// TIA Portal V16 export
// export: Created 2024-06-17T18:37:12.7801223Z, ExportSetting WithDefaults, DisplayName Totally Integrated Automation Portal, DisplayVersion V16, DisplayName TIA Portal Version Control Interface, DisplayVersion V16, DisplayName TIA Portal Openness, DisplayVersion V16, DisplayName STEP 7 Professional, DisplayVersion V16, DisplayName STEP 7 Safety, DisplayVersion V16, DisplayName WinCC Advanced, DisplayVersion V16
TYPE "Axis.RB.Di_PLC.Do"
TITLE = Saídas para robô
// stored: IsFailsafeCompliant false
   STRUCT
      "RB.Gi_PLC.Go_NumProg" : Int;   // Numero Programa
      "RB.Di_PLC.Do16_IniciaProcesso" : Bool;   // Autoriza Número de Programa Processo
      "RB.Di_PLC.Do17_ProgramaOK" : Bool;   // Confirma numero de programa
      "RB.Di_PLC.Do18_MotorOn" : Bool;   // Liga Motores
      "RB.Di_PLC.Do19_MotorOff" : Bool;   // Desliga Motores
      "RB.Di_PLC.Do20_StartRob" : Bool;   // Partida Execução Programa (Play)
      "RB.Di_PLC.Do21_StopRob" : Bool;   // Pausa execução programa (Stop)
      "RB.Di_PLC.Do22_Reserva" : Bool;   // Reserva
      "RB.Di_PLC.Do23_Reserva" : Bool;   // Reserva
      "RB.Di_PLC.Do24_CicloVazio" : Bool;   // Modo Ciclo Vazio
      "RB.Di_PLC.Do25_SolicitaParada" : Bool;   // Pedido de Parada para Entrada na Célula
      "RB.Di_PLC.Do26_CancelaTrabalho" : Bool;   // Aborta uma Trajetória Não Iniciada
      "RB.Di_PLC.Do27_ResetFalha" : Bool;   // Reset Falha
      "RB.Di_PLC.Do28_RetornaManutencao" : Bool;   // Pedido de Retorno da Posição de Manutenção
      "RB.Di_PLC.Do29_RetornaCalibracao" : Bool;   // Pedido de Retorno da Posição de Calibração
      "RB.Di_PLC.Do30_RetornaSincronismo" : Bool;   // Pedido de Retorno da Posição de Sincronismo
      "RB.Di_PLC.Do31_Reserva" : Bool;   // Reserva
      "RB.Di_PLC.Do32_Pressao_Ar_OK" : Bool;   // Pressão de Ar OK
      "RB.Di_PLC.Do33_Reserva" : Bool;   // Reserva
      "RB.Di_PLC.Do34_Reserva" : Bool;   // Reserva
      "RB.Di_PLC.Do35_Reserva" : Bool;   // Reserva
      "RB.Di_PLC.Do36_Reserva" : Bool;   // Reserva
      "RB.Di_PLC.Do37_Reserva" : Bool;   // Reserva
      "RB.Di_PLC.Do38_Reserva" : Bool;   // Reserva
      "RB.Di_PLC.Do39_Reserva" : Bool;   // Reserva
      "RB.Di_PLC.Do40_Reserva" : Bool;   // Reserva
      "RB.Di_PLC.Do41_Reserva" : Bool;   // Reserva
      "RB.Di_PLC.Do42_Reserva" : Bool;   // Reserva
      "RB.Di_PLC.Do43_Reserva" : Bool;   // Reserva
      "RB.Di_PLC.Do44_Reserva" : Bool;   // Reserva
      "RB.Di_PLC.Do45_Reserva" : Bool;   // Reserva
      "RB.Di_PLC.Do46_Reserva" : Bool;   // Reserva
      "RB.Di_PLC.Do47_Reserva" : Bool;   // Reserva
      "RB.Di_PLC.Do48_Reserva" : Bool;   // Reserva
      "RB.Di_PLC.Do49_Reserva" : Bool;   // Reserva
      "RB.Di_PLC.Do50_Reserva" : Bool;   // Reserva
      "RB.Di_PLC.Do51_Reserva" : Bool;   // Reserva
      "RB.Di_PLC.Do52_Reserva" : Bool;   // Reserva
      "RB.Di_PLC.Do53_Reserva" : Bool;   // Reserva
      "RB.Di_PLC.Do54_Reserva" : Bool;   // Reserva
      "RB.Di_PLC.Do55_Reserva" : Bool;   // Reserva
      "RB.Di_PLC.Do56_Aut.Trabalho_1" : Bool;   // Autoriza Trabalho 1
      "RB.Di_PLC.Do57_Aut.Trabalho_2" : Bool;   // Autoriza Trabalho 2
      "RB.Di_PLC.Do58_Aut.Trabalho_3" : Bool;   // Autoriza Trabalho 3
      "RB.Di_PLC.Do59_Aut.Trabalho_4" : Bool;   // Autoriza Trabalho 4
      "RB.Di_PLC.Do60_Aut.Trabalho_5" : Bool;   // Autoriza Trabalho 5
      "RB.Di_PLC.Do61_Aut.Trabalho_6" : Bool;   // Autoriza Trabalho 6
      "RB.Di_PLC.Do62_Aut.Trabalho_7" : Bool;   // Autoriza Trabalho 7
      "RB.Di_PLC.Do63_Aut.Trabalho_8" : Bool;   // Autoriza Trabalho 8
      "RB.Di_PLC.Do64_Aut.Trabalho_9" : Bool;   // Autoriza Trabalho 9
      "RB.Di_PLC.Do65_Aut.Trabalho_10" : Bool;   // Autoriza Trabalho 10
      "RB.Di_PLC.Do66_Aut.Trabalho_11" : Bool;   // Autoriza Trabalho 11
      "RB.Di_PLC.Do67_Aut.Trabalho_12" : Bool;   // Autoriza Trabalho 12
      "RB.Di_PLC.Do68_Aut.Trabalho_13" : Bool;   // Autoriza Trabalho 13
      "RB.Di_PLC.Do69_Aut.Trabalho_14" : Bool;   // Autoriza Trabalho 14
      "RB.Di_PLC.Do70_Aut.Trabalho_15" : Bool;   // Autoriza Trabalho 15
      "RB.Di_PLC.Do71_Aut.Trabalho_16" : Bool;   // Autoriza Trabalho 16
      "RB.Di_PLC.Do72_Aut.Trabalho_17" : Bool;   // Autoriza Trabalho 17
      "RB.Di_PLC.Do73_Aut.Trabalho_18" : Bool;   // Autoriza Trabalho 18
      "RB.Di_PLC.Do74_Aut.Trabalho_19" : Bool;   // Autoriza Trabalho 19
      "RB.Di_PLC.Do75_Aut.Trabalho_20" : Bool;   // Autoriza Trabalho 20
      "RB.Di_PLC.Do76_Aut.Trabalho_21" : Bool;   // Autoriza Trabalho 21
      "RB.Di_PLC.Do77_Aut.Trabalho_22" : Bool;   // Autoriza Trabalho 22
      "RB.Di_PLC.Do78_Aut.Trabalho_23" : Bool;   // Autoriza Trabalho 23
      "RB.Di_PLC.Do79_Aut.Trabalho_24" : Bool;   // Autoriza Trabalho 24
      "RB.Di_PLC.Do80_Aut.Trabalho_25" : Bool;   // Autoriza Trabalho 25
      "RB.Di_PLC.Do81_Aut.Trabalho_26" : Bool;   // Autoriza Trabalho 26
      "RB.Di_PLC.Do82_Aut.Trabalho_27" : Bool;   // Autoriza Trabalho 27
      "RB.Di_PLC.Do83_Aut.Trabalho_28" : Bool;   // Autoriza Trabalho 28
      "RB.Di_PLC.Do84_Aut.Trabalho_29" : Bool;   // Autoriza Trabalho 29
      "RB.Di_PLC.Do85_Aut.Trabalho_30" : Bool;   // Autoriza Trabalho 30
      "RB.Di_PLC.Do86_Aut.Trabalho_31" : Bool;   // Autoriza Trabalho 31
      "RB.Di_PLC.Do87_Aut.Trabalho_32" : Bool;   // Autoriza Trabalho 32
      "RB.Di_PLC.Do88_Aut.Intertravamento_1" : Bool;   // Autoriza Acesso Área Intertravamento 1
      "RB.Di_PLC.Do89_Aut.Intertravamento_2" : Bool;   // Autoriza Acesso Área Intertravamento 2
      "RB.Di_PLC.Do90_Aut.Intertravamento_3" : Bool;   // Autoriza Acesso Área Intertravamento 3
      "RB.Di_PLC.Do91_Aut.Intertravamento_4" : Bool;   // Autoriza Acesso Área Intertravamento 4
      "RB.Di_PLC.Do92_Aut.Intertravamento_5" : Bool;   // Autoriza Acesso Área Intertravamento 5
      "RB.Di_PLC.Do93_Aut.Intertravamento_6" : Bool;   // Autoriza Acesso Área Intertravamento 6
      "RB.Di_PLC.Do94_Aut.Intertravamento_7" : Bool;   // Autoriza Acesso Área Intertravamento 7
      "RB.Di_PLC.Do95_Aut.Intertravamento_8" : Bool;   // Autoriza Acesso Área Intertravamento 8
      "RB.Di_PLC.Do96_Aut.Intertravamento_9" : Bool;   // Autoriza Acesso Área Intertravamento 9
      "RB.Di_PLC.Do97_Aut.Intertravamento_10" : Bool;   // Autoriza Acesso Área Intertravamento 10
      "RB.Di_PLC.Do98_Aut.Intertravamento_11" : Bool;   // Autoriza Acesso Área Intertravamento 11
      "RB.Di_PLC.Do99_Aut.Intertravamento_12" : Bool;   // Autoriza Acesso Área Intertravamento 12
      "RB.Di_PLC.Do100_Aut.Intertravamento_13" : Bool;   // Autoriza Acesso Área Intertravamento 13
      "RB.Di_PLC.Do101_Aut.Intertravamento_14" : Bool;   // Autoriza Acesso Área Intertravamento 14
      "RB.Di_PLC.Do102_Aut.Intertravamento_15" : Bool;   // Autoriza Acesso Área Intertravamento 15
      "RB.Di_PLC.Do103_Aut.Intertravamento_16" : Bool;   // Autoriza Acesso Área Intertravamento 16
      "RB.Di_PLC.Do104_Aut.Intertravamento_17" : Bool;   // Autoriza Acesso Área Intertravamento 17
      "RB.Di_PLC.Do105_Aut.Intertravamento_18" : Bool;   // Autoriza Acesso Área Intertravamento 18
      "RB.Di_PLC.Do106_Aut.Intertravamento_19" : Bool;   // Autoriza Acesso Área Intertravamento 19
      "RB.Di_PLC.Do107_Aut.Intertravamento_20" : Bool;   // Autoriza Acesso Área Intertravamento 20
      "RB.Di_PLC.Do108_Aut.Intertravamento_21" : Bool;   // Autoriza Acesso Área Intertravamento 21
      "RB.Di_PLC.Do109_Aut.Intertravamento_22" : Bool;   // Autoriza Acesso Área Intertravamento 22
      "RB.Di_PLC.Do110_Aut.Intertravamento_23" : Bool;   // Autoriza Acesso Área Intertravamento 23
      "RB.Di_PLC.Do111_Aut.Intertravamento_24" : Bool;   // Autoriza Acesso Área Intertravamento 24
      "RB.Di_PLC.Do112_Aut.Intertravamento_25" : Bool;   // Autoriza Acesso Área Intertravamento 25
      "RB.Di_PLC.Do113_Aut.Intertravamento_26" : Bool;   // Autoriza Acesso Área Intertravamento 26
      "RB.Di_PLC.Do114_Aut.Intertravamento_27" : Bool;   // Autoriza Acesso Área Intertravamento 27
      "RB.Di_PLC.Do115_Aut.Intertravamento_28" : Bool;   // Autoriza Acesso Área Intertravamento 28
      "RB.Di_PLC.Do116_Aut.Intertravamento_29" : Bool;   // Autoriza Acesso Área Intertravamento 29
      "RB.Di_PLC.Do117_Aut.Intertravamento_30" : Bool;   // Autoriza Acesso Área Intertravamento 30
      "RB.Di_PLC.Do118_Aut.Intertravamento_31" : Bool;   // Autoriza Acesso Área Intertravamento 31
      "RB.Di_PLC.Do119_Aut.Intertravamento_32" : Bool;   // Autoriza Acesso Área Intertravamento 32
      "RB.Di_PLC.Do120_Rec.FimTrabalho_1" : Bool;   // Reconhecimento Fim de Trabalho 1
      "RB.Di_PLC.Do121_Rec.FimTrabalho_2" : Bool;   // Reconhecimento Fim de Trabalho 2
      "RB.Di_PLC.Do122_Rec.FimTrabalho_3" : Bool;   // Reconhecimento Fim de Trabalho 3
      "RB.Di_PLC.Do123_Rec.FimTrabalho_4" : Bool;   // Reconhecimento Fim de Trabalho 4
      "RB.Di_PLC.Do124_Rec.FimTrabalho_5" : Bool;   // Reconhecimento Fim de Trabalho 5
      "RB.Di_PLC.Do125_Rec.FimTrabalho_6" : Bool;   // Reconhecimento Fim de Trabalho 6
      "RB.Di_PLC.Do126_Rec.FimTrabalho_7" : Bool;   // Reconhecimento Fim de Trabalho 7
      "RB.Di_PLC.Do127_Rec.FimTrabalho_8" : Bool;   // Reconhecimento Fim de Trabalho 8
      "RB.Di_PLC.Do128_Rec.FimTrabalho_9" : Bool;   // Reconhecimento Fim de Trabalho 9
      "RB.Di_PLC.Do129_Rec.FimTrabalho_10" : Bool;   // Reconhecimento Fim de Trabalho 10
      "RB.Di_PLC.Do130_Rec.FimTrabalho_11" : Bool;   // Reconhecimento Fim de Trabalho 11
      "RB.Di_PLC.Do131_Rec.FimTrabalho_12" : Bool;   // Reconhecimento Fim de Trabalho 12
      "RB.Di_PLC.Do132_Rec.FimTrabalho_13" : Bool;   // Reconhecimento Fim de Trabalho 13
      "RB.Di_PLC.Do133_Rec.FimTrabalho_14" : Bool;   // Reconhecimento Fim de Trabalho 14
      "RB.Di_PLC.Do134_Rec.FimTrabalho_15" : Bool;   // Reconhecimento Fim de Trabalho 15
      "RB.Di_PLC.Do135_Rec.FimTrabalho_16" : Bool;   // Reconhecimento Fim de Trabalho 16
      "RB.Di_PLC.Do136_Rec.FimTrabalho_17" : Bool;   // Reconhecimento Fim de Trabalho 17
      "RB.Di_PLC.Do137_Rec.FimTrabalho_18" : Bool;   // Reconhecimento Fim de Trabalho 18
      "RB.Di_PLC.Do138_Rec.FimTrabalho_19" : Bool;   // Reconhecimento Fim de Trabalho 19
      "RB.Di_PLC.Do139_Rec.FimTrabalho_20" : Bool;   // Reconhecimento Fim de Trabalho 20
      "RB.Di_PLC.Do140_Rec.FimTrabalho_21" : Bool;   // Reconhecimento Fim de Trabalho 21
      "RB.Di_PLC.Do141_Rec.FimTrabalho_22" : Bool;   // Reconhecimento Fim de Trabalho 22
      "RB.Di_PLC.Do142_Rec.FimTrabalho_23" : Bool;   // Reconhecimento Fim de Trabalho 23
      "RB.Di_PLC.Do143_Rec.FimTrabalho_24" : Bool;   // Reconhecimento Fim de Trabalho 24
      "RB.Di_PLC.Do144_Rec.FimTrabalho_25" : Bool;   // Reconhecimento Fim de Trabalho 25
      "RB.Di_PLC.Do145_Rec.FimTrabalho_26" : Bool;   // Reconhecimento Fim de Trabalho 26
      "RB.Di_PLC.Do146_Rec.FimTrabalho_27" : Bool;   // Reconhecimento Fim de Trabalho 27
      "RB.Di_PLC.Do147_Rec.FimTrabalho_28" : Bool;   // Reconhecimento Fim de Trabalho 28
      "RB.Di_PLC.Do148_Rec.FimTrabalho_29" : Bool;   // Reconhecimento Fim de Trabalho 29
      "RB.Di_PLC.Do149_Rec.FimTrabalho_30" : Bool;   // Reconhecimento Fim de Trabalho 30
      "RB.Di_PLC.Do150_Rec.FimTrabalho_31" : Bool;   // Reconhecimento Fim de Trabalho 31
      "RB.Di_PLC.Do151_Rec.FimTrabalho_32" : Bool;   // Reconhecimento Fim de Trabalho 32
      "RB.Di_PLC.Do152_Fluxo_Agua_Equip_1" : Bool;   // Fluxo de Água OK Equipamento 1
      "RB.Di_PLC.Do153_Fluxo_Agua_Equip_2" : Bool;   // Fluxo de Água OK Equipamento 2
      "RB.Di_PLC.Do154_Fluxo_Agua_Equip_3" : Bool;   // Fluxo de Água OK Equipamento 3
      "RB.Di_PLC.Do155_Fluxo_Agua_Equip_4" : Bool;   // Fluxo de Água OK Equipamento 4
      "RB.Di_PLC.Do156_Fluxo_Agua_Equip_5" : Bool;   // Fluxo de Água OK Equipamento 5
      "RB.Di_PLC.Do157_Fluxo_Agua_Equip_6" : Bool;   // Fluxo de Água OK Equipamento 6
      "RB.Di_PLC.Do158_Fluxo_Agua_Equip_7" : Bool;   // Fluxo de Água OK Equipamento 7
      "RB.Di_PLC.Do159_Fluxo_Agua_Equip_8" : Bool;   // Fluxo de Água OK Equipamento 8
      "RB.Di_PLC.Do160_PnetAtivadaEquip_1" : Bool;   // Rede Profinet Ativada Equipamento 1
      "RB.Di_PLC.Do161_PnetAtivadaEquip_2" : Bool;   // Rede Profinet Ativada Equipamento 2
      "RB.Di_PLC.Do162_PnetAtivadaEquip_3" : Bool;   // Rede Profinet Ativada Equipamento 3
      "RB.Di_PLC.Do163_PnetAtivadaEquip_4" : Bool;   // Rede Profinet Ativada Equipamento 4
      "RB.Di_PLC.Do164_PnetAtivadaEquip_5" : Bool;   // Rede Profinet Ativada Equipamento 5
      "RB.Di_PLC.Do165_PnetAtivadaEquip_6" : Bool;   // Rede Profinet Ativada Equipamento 6
      "RB.Di_PLC.Do166_PnetAtivadaEquip_7" : Bool;   // Rede Profinet Ativada Equipamento 7
      "RB.Di_PLC.Do167_PnetAtivadaEquip_8" : Bool;   // Rede Profinet Ativada Equipamento 8
      "RB.Di_PLC.Do168_PnetDesatEquip_1" : Bool;   // Rede Profinet Desativada Equipamento 1
      "RB.Di_PLC.Do169_PnetDesatEquip_2" : Bool;   // Rede Profinet Desativada Equipamento 2
      "RB.Di_PLC.Do170_PnetDesatEquip_3" : Bool;   // Rede Profinet Desativada Equipamento 3
      "RB.Di_PLC.Do171_PnetDesatEquip_4" : Bool;   // Rede Profinet Desativada Equipamento 4
      "RB.Di_PLC.Do172_PnetDesatEquip_5" : Bool;   // Rede Profinet Desativada Equipamento 5
      "RB.Di_PLC.Do173_PnetDesatEquip_6" : Bool;   // Rede Profinet Desativada Equipamento 6
      "RB.Di_PLC.Do174_PnetDesatEquip_7" : Bool;   // Rede Profinet Desativada Equipamento 7
      "RB.Di_PLC.Do175_PnetDesatEquip_8" : Bool;   // Rede Profinet Desativada Equipamento 8
      "RB.Di_PLC.Do176_RetornaTrEletEquip_1" : Bool;   // Retorna Troca de Eletrodo Equipamento 1
      "RB.Di_PLC.Do177_RetornaTrEletEquip_2" : Bool;   // Retorna Troca de Eletrodo Equipamento 2
      "RB.Di_PLC.Do178_RetornaTrEletEquip_3" : Bool;   // Retorna Troca de Eletrodo Equipamento 3
      "RB.Di_PLC.Do179_RetornaTrEletEquip_4" : Bool;   // Retorna Troca de Eletrodo Equipamento 4
      "RB.Di_PLC.Do180_RetornaTrEletEquip_5" : Bool;   // Retorna Troca de Eletrodo Equipamento 5
      "RB.Di_PLC.Do181_RetornaTrEletEquip_6" : Bool;   // Retorna Troca de Eletrodo Equipamento 6
      "RB.Di_PLC.Do182_RetornaTrEletEquip_7" : Bool;   // Retorna Troca de Eletrodo Equipamento 7
      "RB.Di_PLC.Do183_RetornaTrEletEquip_8" : Bool;   // Retorna Troca de Eletrodo Equipamento 8
      "RB.Di_PLC.Do184_RetornaFresagem_1" : Bool;   // Retorna Fresagem Equipamento 1
      "RB.Di_PLC.Do185_RetornaFresagem_2" : Bool;   // Retorna Fresagem Equipamento 2
      "RB.Di_PLC.Do186_RetornaFresagem_3" : Bool;   // Retorna Fresagem Equipamento 3
      "RB.Di_PLC.Do187_RetornaFresagem_4" : Bool;   // Retorna Fresagem Equipamento 4
      "RB.Di_PLC.Do188_RetornaFresagem_5" : Bool;   // Retorna Fresagem Equipamento 5
      "RB.Di_PLC.Do189_RetornaFresagem_6" : Bool;   // Retorna Fresagem Equipamento 6
      "RB.Di_PLC.Do190_RetornaFresagem_7" : Bool;   // Retorna Fresagem Equipamento 7
      "RB.Di_PLC.Do191_RetornaFresagem_8" : Bool;   // Retorna Fresagem Equipamento 8
      "RB.Di_PLC.Do192_DeslFuncaoEquip_1" : Bool;   // Desliga Função (Solda, cola) Equipamento 1
      "RB.Di_PLC.Do193_DeslFuncaoEquip_2" : Bool;   // Desliga Função (Solda, cola) Equipamento 2
      "RB.Di_PLC.Do194_DeslFuncaoEquip_3" : Bool;   // Desliga Função (Solda, cola) Equipamento 3
      "RB.Di_PLC.Do195_DeslFuncaoEquip_4" : Bool;   // Desliga Função (Solda, cola) Equipamento 4
      "RB.Di_PLC.Do196_DeslFuncaoEquip_5" : Bool;   // Desliga Função (Solda, cola) Equipamento 5
      "RB.Di_PLC.Do197_DeslFuncaoEquip_6" : Bool;   // Desliga Função (Solda, cola) Equipamento 6
      "RB.Di_PLC.Do198_DeslFuncaoEquip_7" : Bool;   // Desliga Função (Solda, cola) Equipamento 7
      "RB.Di_PLC.Do199_DeslFuncaoEquip_8" : Bool;   // Desliga Função (Solda, cola) Equipamento 8
      "RB.Di_PLC.Do200_CodigoDecisao_B0" : Bool;   // Código de Decisão Bit 0
      "RB.Di_PLC.Do201_CodigoDecisao_B1" : Bool;   // Código de Decisão Bit 1
      "RB.Di_PLC.Do202_CodigoDecisao_B2" : Bool;   // Código de Decisão Bit 2
      "RB.Di_PLC.Do203_CodigoDecisao_B3" : Bool;   // Código de Decisão Bit 3
      "RB.Di_PLC.Do204_CodigoDecisao_B4" : Bool;   // Código de Decisão Bit 4
      "RB.Di_PLC.Do205_CodigoDecisao_B5" : Bool;   // Código de Decisão Bit 5
      "RB.Di_PLC.Do206_CodigoDecisao_B6" : Bool;   // Código de Decisão Bit 6
      "RB.Di_PLC.Do207_CodigoDecisao_B7" : Bool;   // Código de Decisão Bit 7
      "RB.Di_PLC.Do208_Reserva" : Bool;   // Reserva
      "RB.Di_PLC.Do209_Reserva" : Bool;   // Reserva
      "RB.Di_PLC.Do210_Reserva" : Bool;   // Reserva
      "RB.Di_PLC.Do211_Reserva" : Bool;   // Reserva
      "RB.Di_PLC.Do212_Reserva" : Bool;   // Reserva
      "RB.Di_PLC.Do213_Reserva" : Bool;   // Reserva
      "RB.Di_PLC.Do214_Reserva" : Bool;   // Reserva
      "RB.Di_PLC.Do215_Reserva" : Bool;   // Reserva
      "RB.Di_PLC.Do216_Sts.Ava_Grupo_A" : Bool;   // Grupo A avançado (equipamento acoplado)
      "RB.Di_PLC.Do217_Sts.Ava_Grupo_B" : Bool;   // Grupo B avançado (equipamento acoplado)
      "RB.Di_PLC.Do218_Sts.Ava_Grupo_C" : Bool;   // Grupo C avançado (equipamento acoplado)
      "RB.Di_PLC.Do219_Sts.Ava_Grupo_D" : Bool;   // Grupo D avançado (equipamento acoplado)
      "RB.Di_PLC.Do220_Sts.Ava_Grupo_E" : Bool;   // Grupo E avançado (equipamento acoplado)
      "RB.Di_PLC.Do221_Sts.Ava_Grupo_F" : Bool;   // Grupo F avançado (equipamento acoplado)
      "RB.Di_PLC.Do222_Sts.Ava_Grupo_G" : Bool;   // Grupo G avançado (equipamento acoplado)
      "RB.Di_PLC.Do223_Sts.Ava_Grupo_H" : Bool;   // Grupo H avançado (equipamento acoplado)
      "RB.Di_PLC.Do224_Sts.Ava_Grupo_I" : Bool;   // Grupo I avançado (equipamento acoplado)
      "RB.Di_PLC.Do225_Sts.Ava_Grupo_J" : Bool;   // Grupo J avançado (equipamento acoplado)
      "RB.Di_PLC.Do226_Sts.Ava_Grupo_K" : Bool;   // Grupo K avançado (equipamento acoplado)
      "RB.Di_PLC.Do227_Sts.Ava_Grupo_L" : Bool;   // Grupo L avançado (equipamento acoplado)
      "RB.Di_PLC.Do228_Sts.Ava_Grupo_M" : Bool;   // Grupo M avançado (equipamento acoplado)
      "RB.Di_PLC.Do229_Sts.Ava_Grupo_N" : Bool;   // Grupo N avançado (equipamento acoplado)
      "RB.Di_PLC.Do230_Sts.Ava_Grupo_O" : Bool;   // Grupo O avançado (equipamento acoplado)
      "RB.Di_PLC.Do231_Sts.Ava_Grupo_P" : Bool;   // Grupo P avançado (equipamento acoplado)
      "RB.Di_PLC.Do232_Sts.Rec_Grupo_A" : Bool;   // Grupo A Recuado (equipamento acoplado)
      "RB.Di_PLC.Do233_Sts.Rec_Grupo_B" : Bool;   // Grupo B Recuado (equipamento acoplado)
      "RB.Di_PLC.Do234_Sts.Rec_Grupo_C" : Bool;   // Grupo C Recuado (equipamento acoplado)
      "RB.Di_PLC.Do235_Sts.Rec_Grupo_D" : Bool;   // Grupo D Recuado (equipamento acoplado)
      "RB.Di_PLC.Do236_Sts.Rec_Grupo_E" : Bool;   // Grupo E Recuado (equipamento acoplado)
      "RB.Di_PLC.Do237_Sts.Rec_Grupo_F" : Bool;   // Grupo F Recuado (equipamento acoplado)
      "RB.Di_PLC.Do238_Sts.Rec_Grupo_G" : Bool;   // Grupo G Recuado (equipamento acoplado)
      "RB.Di_PLC.Do239_Sts.Rec_Grupo_H" : Bool;   // Grupo H Recuado (equipamento acoplado)
      "RB.Di_PLC.Do240_Sts.Rec_Grupo_I" : Bool;   // Grupo I Recuado (equipamento acoplado)
      "RB.Di_PLC.Do241_Sts.Rec_Grupo_J" : Bool;   // Grupo J Recuado (equipamento acoplado)
      "RB.Di_PLC.Do242_Sts.Rec_Grupo_K" : Bool;   // Grupo K Recuado (equipamento acoplado)
      "RB.Di_PLC.Do243_Sts.Rec_Grupo_L" : Bool;   // Grupo L Recuado (equipamento acoplado)
      "RB.Di_PLC.Do244_Sts.Rec_Grupo_M" : Bool;   // Grupo M Recuado (equipamento acoplado)
      "RB.Di_PLC.Do245_Sts.Rec_Grupo_N" : Bool;   // Grupo N Recuado (equipamento acoplado)
      "RB.Di_PLC.Do246_Sts.Rec_Grupo_O" : Bool;   // Grupo O Recuado (equipamento acoplado)
      "RB.Di_PLC.Do247_Sts.Rec_Grupo_P" : Bool;   // Grupo P Recuado (equipamento acoplado)
      "RB.Di_PLC.Do248_FimMovimentoDisp_1" : Bool;   // Dispositivo: Fim Movimento Requisitado 1
      "RB.Di_PLC.Do249_FimMovimentoDisp_2" : Bool;   // Dispositivo: Fim Movimento Requisitado 2
      "RB.Di_PLC.Do250_FimMovimentoDisp_3" : Bool;   // Dispositivo: Fim Movimento Requisitado 3
      "RB.Di_PLC.Do251_FimMovimentoDisp_4" : Bool;   // Dispositivo: Fim Movimento Requisitado 4
      "RB.Di_PLC.Do252_FimMovimentoDisp_5" : Bool;   // Dispositivo: Fim Movimento Requisitado 5
      "RB.Di_PLC.Do253_FimMovimentoDisp_6" : Bool;   // Dispositivo: Fim Movimento Requisitado 6
      "RB.Di_PLC.Do254_FimMovimentoDisp_7" : Bool;   // Dispositivo: Fim Movimento Requisitado 7
      "RB.Di_PLC.Do255_FimMovimentoDisp_8" : Bool;   // Dispositivo: Fim Movimento Requisitado 8
   END_STRUCT;
END_TYPE
